Omron Sysmac Studio project Meca500_EtherCAT_Example_6 (Sysmac Studio 1.40.0.64008, StandardProject)

# Controller new_Controller_0: NX1P2-9024DT1 version 1.16
Units and slaves: Node1 : Meca500 (E001)
Task PrimaryTask (priority 4, period or condition 2000): Main

VAR_GLOBAL
    bSTART : BOOL;
    Deactivate : BOOL;  (* at ECAT://node#1/Robot Control_Deactivate_7200_01 *)
    Activate : BOOL;  (* at ECAT://node#1/Robot Control_Activate_7200_02 *)
    Home : BOOL;  (* at ECAT://node#1/Robot Control_Home_7200_03 *)
    SetMoveID : UINT;  (* at ECAT://node#1/Motion Control_Move ID_7310_01 *)
    SetPoint : BOOL;  (* at ECAT://node#1/Motion Control_SetPoint_7310_02 *)
    PauseMove : BOOL;  (* at ECAT://node#1/Motion Control_Pause_7310_03 *)
    ClearMove : BOOL;  (* at ECAT://node#1/Motion Control_Clear Move_7310_04 *)
    MoveCmd : UDINT;  (* at ECAT://node#1/Move_Move Command_7305_00 *)
    MoveArg1 : REAL;  (* at ECAT://node#1/Move_SubIndex 001_7306_01 *)
    MoveArg2 : REAL;  (* at ECAT://node#1/Move_SubIndex 002_7306_02 *)
    MoveArg3 : REAL;  (* at ECAT://node#1/Move_SubIndex 003_7306_03 *)
    MoveArg4 : REAL;  (* at ECAT://node#1/Move_SubIndex 004_7306_04 *)
    MoveArg5 : REAL;  (* at ECAT://node#1/Move_SubIndex 005_7306_05 *)
    MoveArg6 : REAL;  (* at ECAT://node#1/Move_SubIndex 006_7306_06 *)
    isActivated : BOOL;  (* at ECAT://node#1/Robot Status_Activated_6010_03 *)
    isHomed : BOOL;  (* at ECAT://node#1/Robot Status_Homed_6010_04 *)
    GetCheckPoint : UDINT;  (* at ECAT://node#1/Motion Status_CheckPoint_6015_01 *)
    GetMoveID : UINT;  (* at ECAT://node#1/Motion Status_Move ID_6015_02 *)
    isPaused : BOOL;  (* at ECAT://node#1/Motion Status_Paused_6015_04 *)
    isCleared : BOOL;  (* at ECAT://node#1/Motion Status_FIFO Cleared_6015_07 *)
    J1Pose : REAL;  (* at ECAT://node#1/Joint Set_SubIndex 001_6030_01 *)
    J2Pose : REAL;  (* at ECAT://node#1/Joint Set_SubIndex 002_6030_02 *)
    J3Pose : REAL;  (* at ECAT://node#1/Joint Set_SubIndex 003_6030_03 *)
    J4Pose : REAL;  (* at ECAT://node#1/Joint Set_SubIndex 004_6030_04 *)
    J5Pose : REAL;  (* at ECAT://node#1/Joint Set_SubIndex 005_6030_05 *)
    J6Pose : REAL;  (* at ECAT://node#1/Joint Set_SubIndex 006_6030_06 *)
END_VAR

PROGRAM Main
VAR
    nState : UINT := 1;
    nCounter : UINT := 1;
END_VAR
VAR_EXTERNAL
    Activate : BOOL;
    isActivated : BOOL;
    Home : BOOL;
    isHomed : BOOL;
    J1Pose : REAL;
    MoveCmd : UDINT;
    MoveArg1 : REAL;
    MoveArg2 : REAL;
    J2Pose : REAL;
    MoveArg3 : REAL;
    J3Pose : REAL;
    MoveArg4 : REAL;
    J4Pose : REAL;
    MoveArg5 : REAL;
    J5Pose : REAL;
    MoveArg6 : REAL;
    J6Pose : REAL;
    SetPoint : BOOL;
    SetMoveID : UINT;
    GetMoveID : UINT;
    bSTART : BOOL;
    Deactivate : BOOL;
    GetCheckPoint : UDINT;
    isPaused : BOOL;
    isCleared : BOOL;
    PauseMove : BOOL;
    ClearMove : BOOL;
END_VAR
CASE nState OF
		1:	
		nCounter:=1;
		// Activate and Home the Robot
		IF isActivated = TRUE AND isHomed = TRUE THEN
			nState := 2;
		ELSIF isActivated =TRUE THEN
			Home:= TRUE;
		ELSE
			Activate := TRUE;
		END_IF;
		
		2:
		// Set the Joint Velocity
		MoveCmd:= 8;
		MoveArg1:= 20;
		
		// Update the MoveID
		SetMoveID:= nCounter;
		// Set the SetPoint to True to enable sending the command to FIFO command buffer
		SetPoint:= TRUE;
		nState:=3;
		
		3:
		// Set the Cartesian Linear Velocity
		MoveCmd:= 11;
		MoveArg1:= 150;
		// Update the MoveID
		nCounter:=nCounter+1;
		SetMoveID:= nCounter;
		nState:=4;
		
		4:
		// Set Blending
		MoveCmd:= 12;
		MoveArg1:=100;
		// Update the MoveID
		nCounter:=nCounter+1;
		SetMoveID:= nCounter;
		nState:= 5;
		
		5:
		MoveCmd:= 2;
		MoveArg1:= 75;
		MoveArg2:=-150;
		MoveArg3:=150;
		MoveArg4:= 180;
		MoveArg5:= 0;
		MoveArg6:=180;
		// Update the MoveID
		nCounter:=nCounter+1;
		SetMoveID:= nCounter;
		nState:= 6;
		
		6:
		// Set CheckPoint Trigger
		MoveCmd:= 17;
		MoveArg1:= 100;
		// Update the MoveID
		nCounter:=nCounter+1;
		SetMoveID:= nCounter;
		nState:= 7;
		
		7:
		// Wait for the CheckPoint
		IF GetCheckPoint = 100 THEN
			nState:=8;
		END_IF;
		
		8:
		MoveCmd:= 3;
		MoveArg1:= 75;
		MoveArg2:= 150;
		MoveArg3:= 150;
		MoveArg4:= 180;
		MoveArg5:= 0;
		MoveArg6:= 180;
		// Update the MoveID
		nCounter:=nCounter+1;
		SetMoveID:= nCounter;
		nState:= 9;
		
		9:
		MoveCmd:= 3;
		MoveArg1:= 175;
		MoveArg2:= 150;
		MoveArg3:= 150;
		MoveArg4:= 180;
		MoveArg5:= 0;
		MoveArg6:= 180;
		// Update the MoveID
		nCounter:=nCounter+1;
		SetMoveID:= nCounter;
		nState:= 10;
		
		10:
		MoveCmd:= 3;
		MoveArg1:= 175;
		MoveArg2:= -150;
		MoveArg3:= 150;
		MoveArg4:= 180;
		MoveArg5:= 0;
		MoveArg6:= 180;
		// Update the MoveID
		nCounter:=nCounter+1;
		SetMoveID:= nCounter;
		nState:= 11;
		
		11:
		MoveCmd:= 3;
		MoveArg1:= 75;
		MoveArg2:= -150;
		MoveArg3:= 150;
		MoveArg4:= 180;
		MoveArg5:= 0;
		MoveArg6:= 180;
		// Update the MoveID
		nCounter:=nCounter+1;
		SetMoveID:= nCounter;
		nState:= 12;
		
		12:
		MoveCmd:=17;
		MoveArg1:= 200;
		// Update the MoveID
		nCounter:=nCounter+1;
		SetMoveID:= nCounter;
		nState:= 13;		
		
		13:
		// Wait for the CheckPoint
		IF GetCheckPoint = 200 THEN
			nState:= 5;
		END_IF;
						
	END_CASE;
END_PROGRAM